TYPE Weight : (Empty, Light, Heavy);
END_TYPE;

(* stored: Version 1.1.0.1
   DUT Weight: Id {55b6e378-65c8-43c8-8912-8c46830356b4} *)
